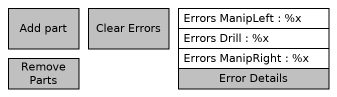
rounded rectangle at (0,0)-(71,41): text "Add part"; alarm colour if PRG_Simulator.bAddPartOnConvIn; taps PRG_Simulator.bAddPartOnConvIn
rounded rectangle at (80,0)-(161,41): text "Clear Errors"; alarm colour if PRG_Simulator.bClearErrors; taps PRG_Simulator.bClearErrors
rectangle at (170,0)-(321,21): text "Errors ManipLeft : %x"; shows PRG_Simulator.wError_ManipL; alarm colour if PRG_Simulator.wError_ManipL > 0
rounded rectangle at (0,50)-(71,81): text "Remove / Parts"; alarm colour if PRG_Simulator.bClearSystem; taps PRG_Simulator.bClearSystem
rectangle at (170,20)-(321,41): text "Errors Drill : %x"; shows PRG_Simulator.wError_Drill; alarm colour if PRG_Simulator.wError_Drill > 0
rectangle at (170,40)-(321,61): text "Errors ManipRight : %x"; shows PRG_Simulator.wError_ManipR; alarm colour if PRG_Simulator.wError_ManipR > 0
rounded rectangle at (170,60)-(321,81): text "Error Details"; opens VC_ErrorDetails
*)

(* Visualisation Simulator/VISU_SimulatedMachine
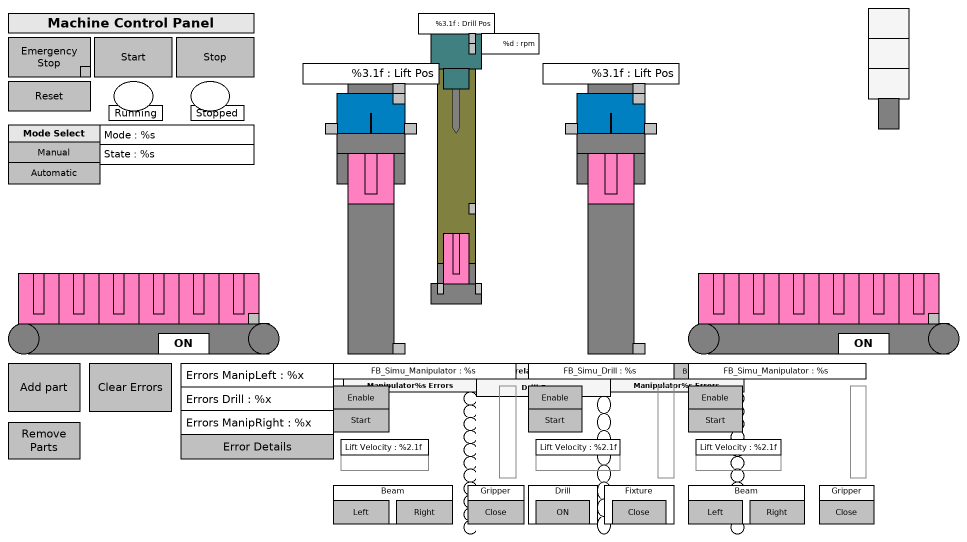
embedded screen at (335,320)-(736,491): VC_ErrorDetails
embedded screen at (0,-30)-(246,141): VC_Panel_MachineControl
embedded screen at (410,-30)-(531,261): VC_Simu_Drill
embedded screen at (0,230)-(271,311): VC_Simu_Conv_In
embedded screen at (0,320)-(326,416): VC_SimuMach_Controls
embedded screen at (325,320)-(516,481): VC_FB_Simu_Manipulator
embedded screen at (250,10)-(431,311): VC_Simu_Manipulator
embedded screen at (490,10)-(671,311): VC_Simu_Manipulator
embedded screen at (680,320)-(866,481): VC_FB_Simu_Manipulator
embedded screen at (520,320)-(666,481): VC_FB_Simu_Drill
embedded screen at (680,230)-(951,311): VC_Simu_Conv_In
embedded screen at (860,-35)-(901,86): VC_Beacon
*)
